FUNCTION_BLOCK BraAttHa
VAR_INPUT
END_VAR
VAR_OUTPUT
END_VAR
VAR
	//eWriteState: (FILE_OPEN_TRIGGER,FILE_OPEN, WAIT_FOR_EVENT, WRITE_EVENT_TRIGGER,WRITE_EVENT, FILE_CLOSE_TRIGGER, FILE_CLOSE, ERROR);
	
END_VAR

END_FUNCTION_BLOCK

(* stored: Version 1.1.0.1, ProductVersion 3.1.4024.12
   POU BraAttHa: Id {de115610-19ec-4aec-809c-058bd69aa67c}, SpecialFunc None *)
